FUNCTION_BLOCK MemoryLogger IMPLEMENTS EventLogger
VAR_INPUT
END_VAR
VAR_OUTPUT
END_VAR
VAR
  event_history: ARRAY[1..Properties.NUM_EVENT_HISTORY] OF EventMessage;
END_VAR

METHOD submit_event_message
VAR_INPUT
	ev: EventMessage;
END_VAR
F_FIFO_WRITE(SIZEOF(ev), ADR(ev), SIZEOF(event_history), ADR(event_history));
END_METHOD

END_FUNCTION_BLOCK

(* stored: Version 1.1.0.1, ProductVersion 3.1.4024.9
   POU MemoryLogger: Id {96136309-a53e-49de-920d-d5f50ab34f7f}, SpecialFunc None
   Method submit_event_message: Id {e515f482-fb51-429d-880d-23c8a80c9002} *)
